FUNCTION F_RolDownTime : TOD
VAR_INPUT
	rSunRise			: REAL;
	todRef				: TOD; (* mittlere Referenzzeit *)
	dwMinFact_neg	: DWORD;
	dwMinFact_pos	: DWORD;
END_VAR
VAR
	dwDate 		: DWORD;
	dwTodRef 	: DWORD;
	rTodRef 	: REAL;
	dwYearDay : DWORD;

	rPi				: REAL;
	rResult		: REAL;
	dwResult	: DWORD;

END_VAR

IF (rSunRise > 0) THEN
	rResult := rSunRise * DWORD_TO_REAL(dwMinFact_pos) * 60000;
ELSE
	rResult := rSunRise * DWORD_TO_REAL(dwMinFact_neg) * 60000;
END_IF

rTodRef := TOD_TO_REAL(todRef);
dwResult := REAL_TO_DWORD(rTodRef + rResult) / 1000 * 1000;

F_RolDownTime := DWORD_TO_TOD(dwResult);

END_FUNCTION

(* stored: Version 1.1.0.1, ProductVersion 3.1.4018.5
   POU F_RolDownTime: Id {c282c80e-87dc-4d47-8e6e-0d5647a66846}, SpecialFunc None *)
